Staubli VAL3: password.pjx

Parameters version=s7.8.3 stackSize=5000 millimeterUnit=true
Program file=start.pgx
Program file=stop.pgx
Data file=password.dtx
